# B&R Automation Studio project Embraco_PracoviskoPopisovaniaLaserom (part 2)

#### Main.st - Init, cyclic, exit code
```iecst
PROGRAM _INIT
	(* Insert code here *)

END_PROGRAM

PROGRAM _CYCLIC
	//0 - 0 - Porucha - nizky tlak vzduchu !!!
	//1 - 1 - Poruchy prepatovej ochrany rozvadzaca !!!
	//2 - 2 - Porucha modulu BC1 - Modul 8DI/DO !!!
	//3 - 3 - Porucha modulu DI1 - Modul 16DI !!!
	//4 - 4 - Porucha modulu SI1 - Modul safety 4SI !!!
	//5 - 5 - Porucha modulu XV1 - Komunikacny modul ventiloveho terminalu !!!
	//6 - 6 - Porucha komunikacie s kamerou !!!
	//7 - 7 - Porucha - bolo stlacene tlacitko CS na paneli zariadenia !!!
	//8 - 8 - Porucha - bolo stlacene tlacitko CS kamery !!!
	//9 - 9 - Porucha napajania odsavania !!!
	//10 - 10 - Porucha napajania lasera !!!
	//11 - 11 - Vstupny oddelovac - porucha zasunutia 1 stopra !!!
	//12 - 12 -  Vstupny oddelovac - porucha zasunutia 2 stopra !!!
	//13 - 13 -  Vstupny oddelovac - porucha vysunutia 1 stopra !!!
	//14 - 14 - Vstupny oddelovac - porucha vysunutia 2 stopra !!!
	//15 - 15 - Popisovanie - porucha vysunutia stopra zdvizky !!!
	//16 - 16 - Popisovanie - porucha zasunutia stopra zdvizky !!!
	//17 - 17 - Popisovanie - porucha vysunutia zdvizky !!!
	//18 - 18 - Popisovanie - porucha zasunutia zdvizky !!!
	//19 - 19 - Kamera - porucha zasunutia 1 stopra !!!
	//20 - 20 - Kamera - porucha zasunutia 2 stopra !!!
	//21 - 21 - Kamera - porucha vysunutia 1 stopra !!!
	//22 - 22 - Kamera - porucha vysunutia 2 stopra !!!
	//23 - 23 - Popisovanie - porucha safety snimaca statora pod laserom !!!
	//24 - 24 - Popisovanie - stator zostal zaseknuty v pozicii popisovania laserom !!!
	//25 - 25 - Popisovanie - laser nieje pripraveny !!!
	//26 - 26 - Popisovanie - porucha odoslania spravy do lasera !!!
	//27 - 27 - Porucha lasera !!!
	//28 - 28 - Porucha kamery !!!
	//29 - 29 - Popisovanie - porucha zvolenia spravy v lasery !!!

	//*********************************Zistenie alarmu************************************************************//
	FOR i:=0 TO 100 BY 1 DO
		Alarmy[i];
		IF Alarmy[i] = TRUE THEN
			NastalaPorucha:= TRUE;
		END_IF
	END_FOR

	//*********************************Blikanie symbolu poruchy na OP*****************************************//
	IF NastalaPorucha THEN
		ZobrazSymbolAlarmu:= Blikac500ms;
	ELSE
		ZobrazSymbolAlarmu:= FALSE;
	END_IF

	//*********************************Zelené svetlo majáka****************************************************//
	IF Zariadenie.STAV.Automat AND NOT Zariadenie.STAV.PoINIT THEN
		Zariadenie.OUT.Majak_ZeleneSvetlo:= Blikac200ms;
	ELSIF Zariadenie.STAV.Automat AND Zariadenie.STAV.PoINIT THEN
		Zariadenie.OUT.Majak_ZeleneSvetlo:= TRUE;
	ELSE
		Zariadenie.OUT.Majak_ZeleneSvetlo:= FALSE;
	END_IF

	//**********************************Žlté svetlo majáka*****************************************************//

	IF Popisovanie.IN.Laser_StavBUSY THEN
		Zariadenie.OUT.Majak_ZlteSvetlo:= TRUE;
	ELSE
		Zariadenie.OUT.Majak_ZlteSvetlo:= FALSE;
	END_IF

	//**********************************Červené svetlo majáka***************************************************//
	IF NastalaPorucha THEN
		Zariadenie.OUT.Majak_CerveneSvetlo:= Blikac200ms;
	ELSE
		Zariadenie.OUT.Majak_CerveneSvetlo:= FALSE;
	END_IF

	//***********************************Zvuková signalizácia majáka*********************************************//
	IF EDGEPOS (NastalaPorucha = TRUE) THEN
		Zariadenie.Hukacka_ON:= TRUE;
	END_IF

	IF Zariadenie.Hukacka_ON THEN
		Zariadenie.OUT.Majak_Hukacka:= Blikac500ms;
	ELSE
		Zariadenie.OUT.Majak_Hukacka:= FALSE;
	END_IF

	IF NOT NastalaPorucha THEN
		Zariadenie.Hukacka_ON:= FALSE;
	ELSIF Zariadenie.Hukacka_OFF THEN
		Zariadenie.Hukacka_ON:= FALSE;
	END_IF

	//*********************************Potvrdenie alarmu**********************************************************//
	IF PotvrdenieAlarmov THEN
		Popisovanie.OUT.Laser_ResetPoruchy:= TRUE;
		brsmemset(ADR(Alarmy),0,SIZEOF(Alarmy));
		NastalaPorucha:= FALSE;
		CasPotvrdeniaAlarmu.IN:= TRUE;
		PoruchaVstupnehoOddelovaca:= FALSE;
		PoruchaPopisovania:= FALSE;
		PoruchaCheckera:= FALSE;
		Zariadenie.Hukacka_OFF:= TRUE;
		Zariadenie.STAV.PrebiehaResetPoruchy:= TRUE;
		PotvrdenieAlarmov:= FALSE;
	END_IF

	IF CasPotvrdeniaAlarmu.Q AND NOT Popisovanie.IN.Laser_ALARM THEN
		Popisovanie.OUT.Laser_ResetPoruchy:= FALSE;
		Zariadenie.STAV.PrebiehaResetPoruchy:= FALSE;
		Zariadenie.Hukacka_OFF:= FALSE;
		CasPotvrdeniaAlarmu.IN:= FALSE;
	END_IF

	CasPotvrdeniaAlarmu.PT:= T#2s;
	CasPotvrdeniaAlarmu();

	//******************************Porucha tlaku vzduchu*********************************************************//

	CasMeraniaTlakuVzduchu.IN:= NOT Zariadenie.IN.TlakVzduchu_OK;

	IF CasMeraniaTlakuVzduchu.Q THEN
		Alarmy[0]:= TRUE;
		Zariadenie.Reset:= TRUE;
	END_IF

	CasMeraniaTlakuVzduchu.PT:= T#5s;
	CasMeraniaTlakuVzduchu();

	//*****************************Porucha prepatovej ochrany******************************************************//
	IF Safety.STAV.SafetyPLC_Nabehlo AND NOT Zariadenie.IN.PrepatovaOchrana_OK THEN
		Alarmy[1]:= TRUE;
	END_IF

	//*****************************Porucha modulu BC1***********************************************************//
	IF Safety.STAV.SafetyPLC_Nabehlo AND NOT Zariadenie.STAV.KOM_Modul_BC1_OK THEN
		Alarmy[2]:= TRUE;
		Zariadenie.Reset:= TRUE;
	END_IF

	//*****************************Porucha modulu DI1***********************************************************//
	IF Safety.STAV.SafetyPLC_Nabehlo AND NOT Zariadenie.STAV.KOM_Modul_DI1_OK THEN
		Alarmy[3]:= TRUE;
		Zariadenie.Reset:= TRUE;
	END_IF

	//*****************************Porucha modulu SI1***********************************************************//
	IF Safety.STAV.SafetyPLC_Nabehlo AND NOT Zariadenie.STAV.KOM_Modul_SI1_OK THEN
		Alarmy[4]:= TRUE;
		Zariadenie.Reset:= TRUE;
	END_IF

	//*****************************Porucha modulu XV1***********************************************************//
	CasMeraniaModuluXV1.IN:= Safety.STAV.ZonaCS_Aktivna AND NOT Zariadenie.STAV.KOM_Modul_XV_OK;

	IF CasMeraniaModuluXV1.Q THEN
		Alarmy[5]:= TRUE;
		Zariadenie.Reset:= TRUE;
	END_IF

	CasMeraniaModuluXV1.PT:= T#10s;
	CasMeraniaModuluXV1();

	//*****************************Porucha komunikacie s kamerou***********************************************//
	IF Zariadenie.STAV.Automat AND NOT Zariadenie.STAV.KOM_Checker_OK THEN
		Alarmy[6]:= TRUE;
		Zariadenie.Reset:= TRUE;
	END_IF

	//******************************Bolo stlačené tlačítko CS na ovládacom paneli zariadenia*****************************************************//
	IF EDGENEG (Safety.STAV.CS_Panel_Odblokov) THEN
		Alarmy[7]:= TRUE;
		Zariadenie.Reset:= TRUE;
	END_IF

	//******************************Bolo stlačené tlačítko CS na kamere*****************************************************//
	IF EDGENEG (Safety.STAV.CS_Checker_Odblokov) THEN
		Alarmy[8]:= TRUE;
		Zariadenie.Reset:= TRUE;
	END_IF

	//******************************Porucha napájania odsávania************************************************//
	IF (Zariadenie.STAV.Automat OR Zariadenie.STAV.Manual) AND NOT Zariadenie.IN.NapajanieOdsavania_OK THEN
		Alarmy[9]:= TRUE;
		Zariadenie.Reset:= TRUE;
	END_IF

	//******************************Porucha napájania lasera************************************************//
	IF (Zariadenie.STAV.Automat OR Zariadenie.STAV.Manual) AND NOT Zariadenie.IN.NapajanieLasera_OK THEN
		Alarmy[10]:= TRUE;
		Zariadenie.Reset:= TRUE;
	END_IF

	//******************************Porucha lasera**********************************************************//
//	IF (Zariadenie.STAV.Automat OR Zariadenie.STAV.Manual) AND Popisovanie.IN.Laser_ALARM THEN
//		Alarmy[27]:= TRUE;
//		Zariadenie.Reset:= TRUE;
//	END_IF

	//Tlačítko Reset CS//
	IF Safety.STAV.CS_Checker_Odblokov AND Safety.STAV.CS_Panel_Odblokov AND NOT Safety.STAV.ZonaCS_Aktivna THEN
		Zariadenie.OUT.LED_Tlacitka_RESET_CS:= Blikac500ms;
	ELSIF Safety.STAV.ZonaCS_Aktivna THEN
		Zariadenie.OUT.LED_Tlacitka_RESET_CS:= TRUE;
	ELSE
		Zariadenie.OUT.LED_Tlacitka_RESET_CS:= FALSE;
	END_IF

	//Tlačítko Štart Automat//
	IF NOT Zariadenie.STAV.Automat AND Safety.STAV.ZonaCS_Aktivna AND NOT NastalaPorucha AND Safety.STAV.ZonaVnutroBunky_Aktivna AND NOT Zariadenie.STAV.UkoncenieCyklu AND Zariadenie.IN.TlakVzduchu_OK AND Zariadenie.STAV.Moduly_OK AND Vizu.CisloAktualnejObrazovky = 2 AND NOT Zariadenie.STAV.NezvolenaReceptura AND NOT Zariadenie.KoniecModelu THEN
		Zariadenie.OUT.LED_Dvojtlacitka_StartStop:= Blikac500ms;
	ELSIF Zariadenie.STAV.Automat AND Zariadenie.STAV.UkoncenieCyklu THEN
		Zariadenie.OUT.LED_Dvojtlacitka_StartStop:= Blikac200ms;
	ELSIF Zariadenie.STAV.Automat AND NOT Zariadenie.STAV.PoINIT THEN
		Zariadenie.OUT.LED_Dvojtlacitka_StartStop:= TRUE;
	ELSIF Zariadenie.STAV.Automat AND Zariadenie.STAV.PoINIT THEN
		Zariadenie.OUT.LED_Dvojtlacitka_StartStop:= TRUE;
	ELSE
		Zariadenie.OUT.LED_Dvojtlacitka_StartStop:= FALSE;
	END_IF

END_PROGRAM

PROGRAM _EXIT
	(* Insert code here *)

END_PROGRAM
```

#### Variables.var - Local variables
```iecst
VAR
	i : INT;
	CasPotvrdeniaAlarmu : TON;
	ZapniHukacku : BOOL;
	CasMeraniaTlakuVzduchu : TON;
	CasMeraniaModuluXV1 : TON;
END_VAR
```

### Program Logical/Program/MeranieTaktime (IEC)

#### Main.st - Init, cyclic, exit code
```iecst
PROGRAM _INIT
	(* Insert code here *)

END_PROGRAM

PROGRAM _CYCLIC

	//Meranie taktime bunky//
	IF Zariadenie.TaktTime_START THEN
		Zariadenie.TaktTime_Milisekundy:= Zariadenie.TaktTime_Milisekundy + 2;//Pretože je v taskovej triede 2ms tak prirátaváme + 2//
		IF Zariadenie.TaktTime_Milisekundy >= 1000 THEN
			Zariadenie.TaktTime_Sekundy:= Zariadenie.TaktTime_Sekundy + 1;
			Zariadenie.TaktTime_Milisekundy:= 0;
		END_IF
		IF Zariadenie.TaktTime_Sekundy >= 60 THEN
			Zariadenie.TaktTime_Minuty:= Zariadenie.TaktTime_Minuty + 1;
			Zariadenie.TaktTime_Sekundy:= 0;
		END_IF
		IF Zariadenie.TaktTime_Minuty >= 60 THEN
			Zariadenie.TaktTime_Hodiny:= Zariadenie.TaktTime_Hodiny + 1;
			Zariadenie.TaktTime_Minuty:= 0;
		END_IF
		IF Zariadenie.TaktTime_Hodiny >= 24 THEN
			Zariadenie.TaktTime_RESET:= TRUE;
		END_IF
	END_IF

	IF Zariadenie.TaktTime_RESET THEN
		Zariadenie.TaktTime_START:= FALSE;
		Zariadenie.TaktTime_Milisekundy:= 0;
		Zariadenie.TaktTime_Sekundy:= 0;
		Zariadenie.TaktTime_Minuty:= 0;
		Zariadenie.TaktTime_Hodiny:= 0;
		Zariadenie.TaktTime_RESET:= FALSE;
	END_IF

	IF Zariadenie.TaktTime_ZAPIS THEN
		Zariadenie.TaktTime_NameraneHodiny:= Zariadenie.TaktTime_Hodiny;
		Zariadenie.TaktTime_NameraneMinuty:= Zariadenie.TaktTime_Minuty;
		Zariadenie.TaktTime_NameraneSekundy:= Zariadenie.TaktTime_Sekundy;
		Zariadenie.TaktTime_Milisekundy:= 0;
		Zariadenie.TaktTime_Sekundy:= 0;
		Zariadenie.TaktTime_Minuty:= 0;
		Zariadenie.TaktTime_Hodiny:= 0;
		Zariadenie.TaktTime_ZAPIS:= FALSE;
	END_IF

END_PROGRAM

PROGRAM _EXIT
	(* Insert code here *)

END_PROGRAM
```

### Program Logical/Blikace/Blikanie200ms (IEC)

#### Blikanie200ms.st - Init, cyclic, exit code
```iecst
PROGRAM _INIT
	(* Insert code here *)

END_PROGRAM

PROGRAM _CYCLIC

	IF NOT Blikac200ms THEN
		Blikac200ms:= TRUE;
	ELSE
		Blikac200ms:= FALSE;
	END_IF

END_PROGRAM

PROGRAM _EXIT
	(* Insert code here *)

END_PROGRAM
```

### Program Logical/Blikace/Blikanie500ms (IEC)

#### Blikanie500ms.st - Init, cyclic, exit code
```iecst
PROGRAM _INIT
	(* Insert code here *)

END_PROGRAM

PROGRAM _CYCLIC
	IF NOT Blikac500ms THEN
		Blikac500ms:= TRUE;
	ELSE
		Blikac500ms:= FALSE;
	END_IF

END_PROGRAM

PROGRAM _EXIT
	(* Insert code here *)

END_PROGRAM
```

### Program Logical/Blikace/Blikanie5s (IEC)

#### Blikanie5s.st - Init, cyclic, exit code
```iecst
PROGRAM _INIT
	(* Insert code here *)

END_PROGRAM

PROGRAM _CYCLIC
	IF NOT Blikac5s THEN
		Blikac5s:= TRUE;
	ELSE
		Blikac5s:= FALSE;
	END_IF

END_PROGRAM

PROGRAM _EXIT
	(* Insert code here *)

END_PROGRAM
```

### Program Logical/Blikace/Blikanie1s (IEC)

#### Blikanie1s.st - Init, cyclic, exit code
```iecst
PROGRAM _INIT
	(* Insert code here *)

END_PROGRAM

PROGRAM _CYCLIC
	IF NOT Blikac1s THEN
		Blikac1s:= TRUE;
	ELSE
		Blikac1s:= FALSE;
	END_IF

END_PROGRAM

PROGRAM _EXIT
	(* Insert code here *)

END_PROGRAM
```

### Program Logical/HMI/OvladanieGrafiky (IEC)

#### Main.st - Init, cyclic, exit code
```iecst
PROGRAM _INIT
	Vizu.Zobraz_HlasenieVymenaModelu:= 1;
	Vizu.Zobraz_ResetZariadenia:= 1;
	Vizu.Zobraz_HlasenieNaZdvizkeNGkus:= 1;

END_PROGRAM

PROGRAM _CYCLIC

	//Zobrazenie úvodnej obrazovky//
	IF NOT Safety.STAV.SafetyPLC_Nabehlo THEN
		Vizu.CisloZadanejObrazovky:= 0;
		IF EDGEPOS (Blikac500ms = TRUE) THEN
			Vizu.Slider:= Vizu.Slider+1;
			IF Vizu.Slider > 30 THEN
				Vizu.Slider:= 0;
			END_IF
		END_IF
	END_IF

	//Prepnutie na hlavnú obrazovku//
	IF EDGEPOS (Safety.STAV.SafetyPLC_Nabehlo = TRUE) THEN
		Vizu.CisloZadanejObrazovky:= 1;
	END_IF

	//Prepnutie na obrazovku alarmov//
	IF EDGEPOS(NastalaPorucha) THEN
		Vizu.CisloZadanejObrazovky:= 5;
	END_IF

	//******************************************************Podsvietenie tlačítok**********************************************************//
	//Tlačítko zámku dverí s rozvádzačom//
	IF Safety.IN.DvereBunky_AktuatorVzamku AND NOT Safety.STAV.DvereBunky_Zamknute THEN
		Vizu.LED_TlacitkaZamokDveriBunky:= Blikac500ms;
	ELSIF Safety.STAV.DvereBunky_Zamknute THEN
		Vizu.LED_TlacitkaZamokDveriBunky:= 2;
	ELSE
		Vizu.LED_TlacitkaZamokDveriBunky:= 3;
	END_IF

	//****************************************************Zobrazenie hlásení****************************************************************//
	//Zobrazenie hlásenia zámky vyblokované//
	IF Safety.STAV.VyblokovanieZamkov_Aktivne THEN
		Vizu.Zobraz_HlasenieZamkyVyblokovane:= 0;
	ELSE
		Vizu.Zobraz_HlasenieZamkyVyblokovane:= 1;
	END_IF

	//Zobrazenie hlásenia nízky tlak vzduchu//
	IF NOT Zariadenie.IN.TlakVzduchu_OK THEN
		Vizu.Zobraz_HlasenieNizkyTlakVzduchu:= 0;
	ELSE
		Vizu.Zobraz_HlasenieNizkyTlakVzduchu:= 1;
	END_IF

	//Zobrazenie hlásenia nezvolená receptura//
	//Príznak nezvolená receptura//
	IF Zariadenie.STAV.NezvolenaReceptura THEN
		Vizu.Zobraz_HlasenieNezvolenaRecept:= 0;
	ELSE
		Vizu.Zobraz_HlasenieNezvolenaRecept:= 1;
	END_IF

	//Zobrazenie hlásenia na zdvižke je NG kus//
	IF Popisovanie.STAV.Zdvizka_PritomnostNGkusu THEN
		Vizu.Zobraz_HlasenieNaZdvizkeNGkus:= 0;
	ELSE
		Vizu.Zobraz_HlasenieNaZdvizkeNGkus:= 1;
	END_IF

	//Zobrazenie tlačítka OK v hlásení zmena modelu//
	IF Vizu.Zobraz_HlasenieVymenaModelu = 0 AND NOT Zariadenie.STAV.Automat THEN
		Vizu.Zobraz_TlacitkoOK_ZmenaModelu:= 0;
	END_IF
	IF Vizu.Zobraz_HlasenieVymenaModelu = 1 THEN
		Vizu.Zobraz_TlacitkoOK_ZmenaModelu:= 1;
	END_IF

	//****************************************************Zamknutie tlačítok****************************************************************//
	//Zamknutie tlačítka Režim Automat//
	IF NOT Safety.STAV.ZonaCS_Aktivna THEN
		Vizu.ZamkniTlacitkoRezimAutomat:= 1;
	ELSIF NOT Safety.STAV.ZonaVnutroBunky_Aktivna THEN
		Vizu.ZamkniTlacitkoRezimAutomat:= 1;
	ELSE
		Vizu.ZamkniTlacitkoRezimAutomat:= 0;
	END_IF

	//Zamknutie tlačítka Režim Manual//
	IF NOT Safety.STAV.ZonaCS_Aktivna THEN
		Vizu.ZamkniTlacitkoRezimManual:= 1;
	ELSIF NastalaPorucha THEN
		Vizu.ZamkniTlacitkoRezimManual:= 1;
	ELSIF Zariadenie.STAV.Automat THEN
		Vizu.ZamkniTlacitkoRezimManual:= 1;
	ELSIF NOT Zariadenie.IN.TlakVzduchu_OK THEN
		Vizu.ZamkniTlacitkoRezimManual:= 1;
	ELSIF NOT Zariadenie.STAV.Moduly_OK THEN
		Vizu.ZamkniTlacitkoRezimManual:= 1;
	ELSE
		Vizu.ZamkniTlacitkoRezimManual:= 0;
	END_IF

	//Zamknutie tlačítok ovládanie zdvižky//
	IF NOT Safety.STAV.ZonaVnutroBunky_Aktivna THEN
		Vizu.ZamkniTlacitkaOvladaniaZdvizky:= 1;
	ELSE
		Vizu.ZamkniTlacitkaOvladaniaZdvizky:= 0;
	END_IF

	//Zamknutie tlačítok ovládania zámkov dverí//
	IF Zariadenie.STAV.Automat THEN
		Vizu.ZamkniTlacitkoZamokDveriBunky:= 1;
	ELSE
		Vizu.ZamkniTlacitkoZamokDveriBunky:= 0;
	END_IF

	//Zamknutie tlačítka Priechodný režim//
	IF Zariadenie.STAV.Automat THEN
		Vizu.ZamkniTlacitkoPriechodnyRezim:= 1;
	ELSE
		Vizu.ZamkniTlacitkoPriechodnyRezim:= 0;
	END_IF

	//Zamknutie tlačítka Štart popisovania laserom//
	IF NOT Safety.STAV.ZonaLaser_Aktivna THEN
		Vizu.ZamkniTlacitko_StartPopisovania:= 1;
	ELSIF NOT Popisovanie.IN.Laser_StavREADY THEN
		Vizu.ZamkniTlacitko_StartPopisovania:= 1;
	ELSE
		Vizu.ZamkniTlacitko_StartPopisovania:= 0;
	END_IF

	//Zamknutie tlačítka Laser - výber správy//
	IF Popisovanie.IN.Laser_StavREADY THEN
		Vizu.ZamkniTlacitkoLaserVolbaSpravy:= 0;
	ELSE
		Vizu.ZamkniTlacitkoLaserVolbaSpravy:= 1;
	END_IF

	//Zamknutie tlačítka Laser - poslanie dát správy//
	IF Popisovanie.IN.Laser_StavREADY AND Laser.Status.VyberSpravy_OK THEN
		Vizu.ZamkniTlacitkoLaserPosliData:= 0;
	ELSE
		Vizu.ZamkniTlacitkoLaserPosliData:= 1;
	END_IF

END_PROGRAM

PROGRAM _EXIT
	(* Insert code here *)

END_PROGRAM
```

- Visualisation Logical/HMI/Visu (not shown)

### Program Logical/Komunikacia_Laser/Vycitanie_casu (IEC)

#### citanie_casu_z_PLC.ab - Init, cyclic, exit code
```automation-basic
PROGRAM _INIT
	Zapnutie_citania_casu:=1;

END_PROGRAM

PROGRAM _CYCLIC
	DTStructureGetTime(Zapnutie_citania_casu, ADR(System_Cas_Datum), Status_citania_casu);

	Systemovy_Cas.Hodina:= System_Cas_Datum.hour;
	Systemovy_Cas.Minuta:= System_Cas_Datum.minute;
	Systemovy_Cas.Sekunda:= System_Cas_Datum.second;

	Systemovy_Datum.Den:= System_Cas_Datum.day;
	Systemovy_Datum.Mesiac:= System_Cas_Datum.month;
	Systemovy_Datum.Rok:= System_Cas_Datum.year;

END_PROGRAM

PROGRAM _EXIT
	(* Insert code here *)

END_PROGRAM
```

### Program Logical/Komunikacia_Laser/EthernetovaKomunikacia (IEC)

#### Main.st - Init, cyclic, exit code
```iecst
PROGRAM _INIT
	(* Insert code here *)

END_PROGRAM

PROGRAM _CYCLIC

	Laser_Sprava;

	CASE Client.sStep OF

		0://Čakanie na spustenie komunikácie z laserom//
			IF Laser.Commands.VyberSpravuLasera THEN
				Laser.Status.PoruchaOtvoreniaKomunikacie:= FALSE;
				Laser.Status.PoruchaSpojenia_s_Laserom:= FALSE;
				Laser.Status.PoruchaOdoslaniaDat:= FALSE;
				Laser.Status.PoruchaZatvoreniaKomunikacie:= FALSE;
				Laser.Status.PoruchaPrijatiaDat:= FALSE;
				Laser.Status.VyberSpravy_NG:= FALSE;
				Laser.Status.VyberSpravy_OK:= FALSE;
				Laser.Status.StrataKomunikacie:= FALSE;
				brsmemset(ADR(Laser_Sprava),0,SIZEOF(Laser_Sprava));
				brsmemset(ADR(Laser_Odpoved),0,SIZEOF(Laser_Odpoved));
				brsmemcpy(ADR(Laser_Sprava[0]),ADR(Laser_NazovSpravy),SIZEOF(Laser_NazovSpravy));
				Client.sStep := 1;
			ELSIF Laser.Commands.OdosliDataSpravy THEN
				Laser.Status.PoruchaOtvoreniaKomunikacie:= FALSE;
				Laser.Status.PoruchaSpojenia_s_Laserom:= FALSE;
				Laser.Status.PoruchaOdoslaniaDat:= FALSE;
				Laser.Status.PoruchaZatvoreniaKomunikacie:= FALSE;
				Laser.Status.PoruchaPrijatiaDat:= FALSE;
				Laser.Status.OdoslanieDatSpravy_OK:= FALSE;
				Laser.Status.OdoslanieDatSpravy_NG:= FALSE;
				Laser.Status.StrataKomunikacie:= FALSE;
				brsmemset(ADR(Laser_Sprava),0,SIZEOF(Laser_Sprava));
				brsmemset(ADR(Laser_Odpoved),0,SIZEOF(Laser_Odpoved));
				brsmemcpy(ADR(Laser_Sprava[0]),ADR(Laser_DataSpravy),SIZEOF(Laser_DataSpravy));
				Client.sStep := 1;
			END_IF

		1: //Otvorenie ethernetovej komunikácie//
			Client.TcpOpen_0.enable := 1;
			Client.TcpOpen_0.pIfAddr := 0;  (* Which Interface to open *)
			Client.TcpOpen_0.port := 3490;  (* Port komunikácie s laserom *)
			Client.TcpOpen_0.options := 0;
			Client.TcpOpen_0;  (* Call the Function *)

			IF Client.TcpOpen_0.status = 0 THEN  (* TCP port je otvorený *)
				Client.TcpOpen_timeout := 0;
				Client.sStep := 5;
			ELSIF Client.TcpOpen_0.status = ERR_FUB_BUSY THEN  (* TCP port sa otvára *)
				Client.TcpOpen_timeout := Client.TcpOpen_timeout + 1;
				IF Client.TcpOpen_timeout > 50 THEN
					Laser.Status.PoruchaOtvoreniaKomunikacie:= TRUE;
					Client.TcpOpen_timeout := 0;
					Client.sStep := 100;
				END_IF
				(* Busy *)
			ELSE  (* Goto Error Step *)
				Laser.Status.PoruchaOtvoreniaKomunikacie:= TRUE;
				Client.TcpOpen_timeout := 0;
				Client.sStep := 100;
			END_IF

		5:
			Client.linger_opt.lLinger := 0; (* linger Time = 0 *)
			Client.linger_opt.lOnOff := 1; (* linger Option ON *)
			Client.TcpIoctl_0.enable := 1;
			Client.TcpIoctl_0.ident := Client.TcpOpen_0.ident; (* Connection Ident from AsTP.TCP_Open *)
			Client.TcpIoctl_0.ioctl := tcpSO_LINGER_SET; (* Set Linger Options *)
			Client.TcpIoctl_0.pData := ADR(Client.linger_opt);
			Client.TcpIoctl_0.datalen := SIZEOF(Client.linger_opt);
			Client.TcpIoctl_0;

			IF Client.TcpIoctl_0.status = 0 THEN  (* TcpIoctl successfull *)
				Client.sStep := 10;
			ELSIF Client.TcpIoctl_0.status = ERR_FUB_BUSY THEN  (* TcpIoctl not finished -> redo *)
				(* Busy *)
			ELSE  (* Goto Error Step *)
				Client.sStep := 100;
			END_IF

		10: //Spojenie s laserom//
			Client.TcpClient_0.enable := 1;
			Client.TcpClient_0.ident := Client.TcpOpen_0.ident;  (* Connection Ident from AsTCP.TCP_Open *)
			Client.TcpClient_0.portserv := 3490;  (* Port komunikácie s laserom *)
			Client.TcpClient_0.pServer := ADR('192.168.1.4');  (* Adresa lasera *)
			Client.TcpClient_0;  (* Call the Function*)

			IF Client.TcpClient_0.status = 0 THEN  (* Open ok -> Send Data *)
				Client.TcpClient_timeout := 0;
				Client.sStep := 20;
			ELSIF Client.TcpClient_0.status = ERR_FUB_BUSY THEN  (* TcpClient not finished -> redo *)
				Client.TcpClient_timeout := Client.TcpClient_timeout + 1;
				IF Client.TcpClient_timeout > 50 THEN
					Laser.Status.StrataKomunikacie:= TRUE;
					Client.TcpClient_timeout := 0;
					Client.sStep := 40;
				END_IF

				(* Busy *)
			ELSIF Client.TcpClient_0.status = tcpERR_INVALID THEN  (* Port error -> Close actual connection, and reopen a new one *)
				Client.TcpClient_timeout := 0;
				Client.sStep := 40;
			ELSE  (* Goto Error Step *)
				Laser.Status.PoruchaSpojenia_s_Laserom:= TRUE;
				Client.TcpClient_timeout := 0;
				Client.sStep := 100;
			END_IF

		20: //Poslanie dát do lasera//
			Client.TcpSend_0.enable := 1;
			Client.TcpSend_0.ident := Client.TcpOpen_0.ident;  (* Connection Ident from AsTCP.TCP_Open *)
			Client.TcpSend_0.pData := ADR(Laser_Sprava);  (* Dáta poslané do lasera *)
			Client.TcpSend_0.datalen := SIZEOF(Laser_Sprava);  (* Lenght of data to send *)
			Client.TcpSend_0.flags := 0;
			Client.TcpSend_0;  (* Call the Function*)

			IF Client.TcpSend_0.status = 0 THEN  (* Data was sent sucessfully -> receive data *)
				Client.sStep := 30;
			ELSIF Client.TcpSend_0.status = ERR_FUB_BUSY THEN  (* TcpSend not finished -> redo *)
				(* Busy *)
			ELSIF (Client.TcpSend_0.status = tcpERR_SENTLEN) OR (Client.TcpSend_0.status = tcpERR_NOT_CONNECTED) THEN (* Connection Lost *)
				Laser.Status.StrataKomunikacie:= TRUE;
				Client.sStep := 40;
			ELSE  (* Goto Error Step *)
				Laser.Status.PoruchaOdoslaniaDat:= TRUE;
				Client.sStep := 100;
			END_IF

		30: //Prijatie odpovede s lasera//
			Client.TcpRecv_0.enable := 1;
			Client.TcpRecv_0.ident := Client.TcpOpen_0.ident;  (* Connection Ident from AsTCP.TCP_Open *)
			Client.TcpRecv_0.pData	:= ADR(Laser_Odpoved);  (* Dáta poslané z lasera *)
			Client.TcpRecv_0.datamax := SIZEOF(Laser_Odpoved);  (* Lenght of data buffer *)
			Client.TcpRecv_0.flags := 0;
			Client.TcpRecv_0;  (* Call the Function*)

			IF Client.TcpRecv_0.status = 0 THEN  (* Data was received sucessfully -> Send next packet *)
				Client.recv_timeout := 0;
				Client.sStep := 40;
			ELSIF Client.TcpRecv_0.status = tcpERR_NO_DATA THEN  (* No data received - wait *)
				Client.recv_timeout := Client.recv_timeout + 1;
				IF Client.recv_timeout > 50 THEN
					Client.recv_timeout := 0;
					Laser.Status.PoruchaPrijatiaDat:= TRUE;
					Client.sStep := 40;
				END_IF
				(* No Data received *)
			ELSIF Client.TcpRecv_0.status = ERR_FUB_BUSY THEN  (* TcpRecv not finished -> redo *)
				(* Busy *)
			ELSIF Client.TcpRecv_0.status = tcpERR_NOT_CONNECTED THEN (* Connection Lost *)
				Client.recv_timeout := 0;
				Laser.Status.StrataKomunikacie:= TRUE;
				Client.sStep := 40;
			ELSE  (* Goto Error Step *)
				Laser.Status.PoruchaPrijatiaDat:= TRUE;
				Client.recv_timeout := 0;
				Client.sStep := 100;
			END_IF

		40: //Zatvorenie ethernetovej komunikácie//
			Client.TcpClose_0.enable := 1;
			Client.TcpClose_0.ident := Client.TcpOpen_0.ident;  (* Connection Ident from AsTCP.TCP_Open *)
			Client.TcpClose_0.how := 0;
			Client.TcpClose_0;  (* Call the Function*)

			IF Client.TcpClose_0.status = 0 THEN  (* Close sucessfull -> Reopen the interface *)
				Client.sStep := 50;
			ELSIF Client.TcpClose_0.status = ERR_FUB_BUSY THEN  (* TcpClose not finished -> redo *)
				(* Busy *)
			ELSE  (* Goto Error Step *)
				Laser.Status.PoruchaZatvoreniaKomunikacie:= TRUE;
				Client.sStep := 100;
			END_IF

		50: //Kontrola odpovede z lasera//
			//Ak je status 0 tak je odpoved lasera OK//
			IF Laser.Commands.VyberSpravuLasera THEN
				Laser.Status.VysledokPorovnaniaOdpovede:= brsmemcmp(ADR(Laser_Odpoved),ADR(OK_OdpovedNaVyberSpravy),SIZEOF(OK_OdpovedNaVyberSpravy));
				IF Laser.Status.VysledokPorovnaniaOdpovede = 0 THEN
					Laser.Status.VyberSpravy_OK:= TRUE;
					Laser.Commands.VyberSpravuLasera:= FALSE;
					Client.sStep := 0;
				ELSE
					Laser.Status.VyberSpravy_NG:= TRUE;
					Laser.Commands.VyberSpravuLasera:= FALSE;
					Client.sStep := 0;
				END_IF
			ELSIF Laser.Commands.OdosliDataSpravy THEN
				Laser.Status.VysledokPorovnaniaOdpovede:= brsmemcmp(ADR(Laser_Odpoved),ADR(OK_OdpovedNaDataSpravy),SIZEOF(OK_OdpovedNaDataSpravy));
				IF Laser.Status.VysledokPorovnaniaOdpovede = 0 THEN
					Laser.Status.OdoslanieDatSpravy_OK:= TRUE;
					Laser.Commands.OdosliDataSpravy:= FALSE;
					Client.sStep := 0;
				ELSE
					Laser.Status.OdoslanieDatSpravy_NG:= TRUE;
					Laser.Commands.OdosliDataSpravy:= FALSE;
					Client.sStep := 0;
				END_IF
			END_IF

		100: //Ukončenie komunikácie s laserom//
			Laser.Commands.VyberSpravuLasera:= FALSE;
			Laser.Commands.OdosliDataSpravy:= FALSE;
			Client.sStep := 0;

	END_CASE

END_PROGRAM

PROGRAM _EXIT
	(* Insert code here *)

END_PROGRAM
```

### Program Logical/Komunikacia_Checker/CheckerKomunikacia (IEC)

#### Main.st - Init, cyclic, exit code
```iecst
PROGRAM _INIT

END_PROGRAM

PROGRAM _CYCLIC

	//Vstupy pre checker KOGNEX//
	Checker.COM.ControlWord.0:= Checker.TRIGER_Enable;
	Checker.COM.ControlWord.1:= Checker.TRIGER;
	Checker.COM.ResultControl.1:= Checker.Vysledok_POTVRDENIE;

	//Výstupy z checkera KOGNEX//
	Checker.STAV.TRIGER_Ready:= Checker.COM.StatusWord.0;
	Checker.STAV.BUSY:= Checker.COM.ResultStatus.0;
	Checker.STAV.Vysledok_READY:= Checker.COM.ResultStatus.3;
	Checker.STAV.Vysledok_OK:= Checker.COM.ResultData.0;
	Checker.STAV.Vysledok_NG:= NOT Checker.COM.ResultData.0;

END_PROGRAM

PROGRAM _EXIT
	(* Insert code here *)

END_PROGRAM
```

### Program Logical/Receptury/Receptury (IEC)

#### Main.st - Init, cyclic, exit code
```iecst
PROGRAM _INIT

END_PROGRAM

PROGRAM _CYCLIC

	//Načítanie receptur pri prvom spustení//
	IF EDGEPOS(Safety.STAV.SafetyPLC_Nabehlo = TRUE) THEN
		MpRecipeXml_0.Load:= TRUE;
	END_IF

	//Načítanie receptur z pamäte//
	IF MpRecipeXml_0.Load AND (MpRecipeXml_0.CommandDone OR MpRecipeXml_0.Error) THEN
		MpRecipeXml_0.Load:= FALSE;
		old_i:= 1;
		i:= 0;
		IndexZoznam:= 0;
	END_IF

	//Konfigurácia receptur//
	MpRecipeXml_0.MpLink:= ADR(gRecipeXmlLink);  //takto sa menuje mapp komponenta v configurating view//
	MpRecipeXml_0.Enable:= TRUE;
	MpRecipeXml_0.Category:= ADR('RECEPTURY');
	MpRecipeXml_0.DeviceName:= ADR('HDD');  //Názov media, kde sa budú receptury ukladat//
	MpRecipeXml_0.FileName:= ADR('UlozeneReceptury'); //Názov súboru do ktorého sa receptúry uložia//
	MpRecipeXml_0();

	MpRecipeRegPar_0.MpLink:= ADR(gRecipeXmlLink);
	MpRecipeRegPar_0.Enable:= TRUE;
	MpRecipeRegPar_0.Category:= ADR('RECEPTURY');
	MpRecipeRegPar_0.PVName:= ADR('Receptura'); //Názov premenné, kde je vytvorená štruktura dat pre receptury//
	MpRecipeRegPar_0();

	//Zobrazenie názvou receptúr//
	FOR IndexZoznam:=0 TO 150 BY 1 DO
		ZoznamReceptur[IndexZoznam]:= Receptura[IndexZoznam].NazovStatora;
	END_FOR

	//Posun indexu//
	IF MoveUP THEN
		IF i< 150 THEN
			i:= i+1;
		END_IF
		MoveUP:= FALSE;
	END_IF

	IF MoveDown THEN
		IF i>0 THEN
			i:= i-1;
		END_IF
		MoveDown:= FALSE;
	END_IF

	//Posun indexu po stranách//
	IF MoveUP_Page THEN
		IF i< (150 - 7) THEN
			i:= i+7;
		END_IF
		MoveUP_Page:= FALSE;
	END_IF

	IF MoveDown_Page THEN
		IF i>(0+7) THEN
			i:= i-7;
		END_IF
		MoveDown_Page:= FALSE;
	END_IF

	//Listovanie v uložených recepturach//
	IF old_i <> i THEN
		NazovStatora:= Receptura[i].NazovStatora;
		BOM_kod_Statora:= Receptura[i].BOM_kod_Statora;
		old_i:= i;
	END_IF

	//Uloženie receptury//
	IF UlozRecepturu THEN
		Receptura[i].NazovStatora:= NazovStatora;
		Receptura[i].BOM_kod_Statora:= BOM_kod_Statora;
		MpRecipeXml_0.Save:= TRUE;
		IF MpRecipeXml_0.CommandDone THEN
			MpRecipeXml_0.Save:= FALSE;
			UlozRecepturu:= FALSE;
		END_IF
	END_IF

	//Načitanie receptur do premenných//
	IF NacitajRecepturu THEN
		ZvolenyNazovStatora:= NazovStatora;
		ZvolenyBOM_kod_Statora:= BOM_kod_Statora;
		NacitajRecepturu:= FALSE;
	END_IF

END_PROGRAM

PROGRAM _EXIT
	(* Insert code here *)

END_PROGRAM
```

#### Variables.var - Local variables
```iecst
VAR
	MpRecipeUI_0 : MpRecipeUI;
	UISetup : MpRecipeUISetupType;
	UIConnect : MpRecipeUIConnectType := (0);
	i : UINT;
	old_i : UINT;
	IndexZoznam : UINT;
	MoveUP : BOOL;
	MoveDown : BOOL;
	MoveUP_Page : BOOL;
	MoveDown_Page : BOOL;
END_VAR
```

### Program Logical/PrihlasovaciSystem/PrihlasovaciSystem (IEC)

#### Main.st - Init, cyclic, exit code
```iecst
PROGRAM _INIT
	MpRecipeXml_1.Load:= TRUE;
	ZvolenyUzivatel:= '';
	ZvolenaUroven:= 0;
	TP_ZobrazPopUpPrihlasenie:=1;

END_PROGRAM

PROGRAM _CYCLIC

	//Volanie funkcie SequenceControl//
	SequenceControl(SC:= SC_Uzivatelia);

	//Načítanie receptur z pamäte//
	IF MpRecipeXml_1.Load AND (MpRecipeXml_1.CommandDone OR MpRecipeXml_1.Error) THEN
		MpRecipeXml_1.Load:= FALSE;
		old_a:= 1;
		i:= 0;
		IndexZoznam:= 0;
	END_IF

	//Konfigurácia receptur//
	MpRecipeXml_1.MpLink:= ADR(gUzivatelXmlLink);  //takto sa menuje mapp komponenta v configurating view//
	MpRecipeXml_1.Enable:= TRUE;
	MpRecipeXml_1.Category:= ADR('UZIVATELIA');
	MpRecipeXml_1.Category:= ADR(strCategory);
	MpRecipeXml_1.DeviceName:= ADR('HDD');  //Názov media, kde sa budú receptury ukladat//
	MpRecipeXml_1.FileName:= ADR('UlozenyUzivatel'); //Názov súboru do ktorého sa receptúry uložia//
	MpRecipeXml_1();

	MpRecipeRegPar_1.MpLink:= ADR(gUzivatelXmlLink);
	MpRecipeRegPar_1.Enable:= TRUE;
	MpRecipeRegPar_1.Category:= ADR('UZIVATELIA');
	MpRecipeRegPar_1.PVName:= ADR('Uzivatel'); //Názov premenné, kde je vytvorená štruktura dat pre receptury//
	MpRecipeRegPar_1();

	//Zobrazenie názvou receptúr//
	FOR IndexZoznam:=0 TO 50 BY 1 DO
		ZoznamUzivatelov[IndexZoznam]:= Uzivatel[IndexZoznam].Meno;
	END_FOR

	//Posun indexu//
	IF MoveUP THEN
		IF i< 50 THEN
			i:= i+1;
		END_IF
		MoveUP:= FALSE;
	END_IF

	IF MoveDown THEN
		IF i>0 THEN
			i:= i-1;
		END_IF
		MoveDown:= FALSE;
	END_IF

	//Listovanie v uložených uživateloch//
	IF old_a <> i AND i >= 0 AND i <= 50 THEN
		MenoUzivatela:= Uzivatel[i].Meno;
		HesloUzivatela:= Uzivatel[i].Heslo;
		UrovenUzivatela:= Uzivatel[i].UrovenUzivatela;
		old_a:= i;
	END_IF

	//Prihlasovanie//
	CASE SC_Uzivatelia.Step OF

		0://Vynulovanie uživatela//
			SC_Uzivatelia.StepName:= '0 - Nulovanie';
			UlozUzivatelov:= FALSE;
			PrihlasUzivatela:= FALSE;
			VymazUzivatela:= FALSE;
			OdhlasUzivatela:= FALSE;
			MpRecipeXml_1.Save:= FALSE;
			b:= 0;
			SC_Uzivatelia.ResetStep:= TRUE;
			SC_Uzivatelia.Step:= 1;

		1://Rozhodnutie o činnosti//
			SC_Uzivatelia.StepName:= '1 - Rozhodnutie o cinnosti';
			IF UlozUzivatelov THEN
				SC_Uzivatelia.Step:= 10;
			ELSIF PrihlasUzivatela THEN
				SC_Uzivatelia.Step:= 20;
			ELSIF OdhlasUzivatela THEN
				SC_Uzivatelia.Step:= 30;
			ELSIF VymazUzivatela THEN
				SC_Uzivatelia.Step:= 40;
			END_IF

		10://Ulozenie uzivatela//
			SC_Uzivatelia.StepName:= '10 - Ulozenie uzivatela';
			Uzivatel[i].Meno:= MenoUzivatela;
			Uzivatel[i].Heslo:= HesloUzivatela;
			Uzivatel[i].UrovenUzivatela:= UrovenUzivatela;
			MpRecipeXml_1.Save:= TRUE;
			IF MpRecipeXml_1.CommandDone THEN
				SC_Uzivatelia.ResetStep:= TRUE;
				SC_Uzivatelia.Step:= 0;
			END_IF

		20://Čakanie na prihlásenie uživatela//
			SC_Uzivatelia.StepName:= '20 - Kontrola prazdneho uzivatela';
			IF ZadaneMenoUzivatela <> '' AND ZadaneHesloUzivatela <> '' THEN
				SC_Uzivatelia.ResetStep:= TRUE;
				SC_Uzivatelia.Step:= 21;
			ELSE
				ZadaneHesloUzivatela:= '';
				SC_Uzivatelia.ResetStep:= TRUE;
				SC_Uzivatelia.Step:= 0;
			END_IF

		21://Kontrola prihláseného uživatela//
			SC_Uzivatelia.StepName:= '21 - Kontrola prihláseného uzivatela';
			IF Uzivatel[b].Meno = ZadaneMenoUzivatela AND Uzivatel[b].Heslo = ZadaneHesloUzivatela THEN
				ZvolenyUzivatel:= Uzivatel[b].Meno;
				ZvolenaUroven:= Uzivatel[b].UrovenUzivatela;
				ZadaneHesloUzivatela:= '';
				TP_ZobrazPopUpPrihlasenie:= 1;
				SC_Uzivatelia.ResetStep:= TRUE;
				SC_Uzivatelia.Step:= 0;
			ELSE
				b:= b + 1;
				IF b = 51 OR b < 0 OR b > 51 THEN
					ZadaneMenoUzivatela:= '';
					ZadaneHesloUzivatela:= '';
					SC_Uzivatelia.ResetStep:= TRUE;
					SC_Uzivatelia.Step:= 0;
				END_IF
			END_IF

		30://Odhlásenie uživatela//
			SC_Uzivatelia.StepName:= '30 - Odhlasenie uzivatela';
			ZvolenyUzivatel:= '';
			ZvolenaUroven:= 0;
			SC_Uzivatelia.ResetStep:= TRUE;
			SC_Uzivatelia.Step:= 0;

		40://Vymazanie uživatela//
			SC_Uzivatelia.StepName:= '40 - Vymazanie uzivatela';
			Uzivatel[i].Meno:= '';
			Uzivatel[i].Heslo:= '';
			Uzivatel[i].UrovenUzivatela:= 0;
			MpRecipeXml_1.Save:= TRUE;
			IF MpRecipeXml_1.CommandDone THEN
				SC_Uzivatelia.ResetStep:= TRUE;
				SC_Uzivatelia.Step:= 0;
			END_IF

	END_CASE

END_PROGRAM

PROGRAM _EXIT
	(* Insert code here *)

END_PROGRAM
```

#### Variables.var - Local variables
```iecst
VAR
	strCategory : STRING[80];
	MpRecipeUI_1 : MpRecipeUI;
	UISetup : MpRecipeUISetupType;
	UIConnect : MpRecipeUIConnectType := (0);
	i : INT := 0;
	a : INT;
	old_a : INT := 0;
	MoveUP : BOOL;
	MoveDown : BOOL;
	IndexZoznam : INT;
	b : INT;
	CasOdhlaseniaUzivatela : TON;
END_VAR
```

### Poznamky.txt
```
Heslo do safety - vlmardo
Heslo HMI: login - admin
		   heslo - vlmardo
Takt time - 7s

Obsah QR kódu:
- BOM materiálu - napr.1355470 z receptury
- Dátum výroby - napr.17042019 z PLC
- Čas výroby - napr.1107;1045 z PLC
- Číslo výr. linky - StatorEM
Vedla kódu posledné štvorčíslie BOM materiálu - napr.5470
Názov statora napr.MAF4578

Názov správy lineem

IP adresa PLC 192.168.1.2
IP adresa HMI 192.168.1.3
IP adresa Lasera 192.168.1.4
KOM port laser 3490

IP adresa Checker 192.168.2.2
```
